// TwinCAT 3 PLC project Abschervorrichtung
// ProgramVersion: 3.1.4026.16
// libraries:
//   Tc2_EtherCAT, * (Beckhoff Automation GmbH)
//   Tc2_Standard, * (Beckhoff Automation GmbH)
//   Tc2_System, * (Beckhoff Automation GmbH)
// project tree:
//   DUTs/ ST_OperatingTime.TcDUT, ST_OpMode.TcDUT (not stored)
//   GVLs/ GVL_CouplerOnDesk.TcGVL (not stored)
//   / PlcTask.TcTTO
//   POUs/ FB_EL6090.TcPOU (not stored), FB_SetOpMode.TcPOU (not stored), F_Convert_to_OperatingTime.TcPOU (not stored), MAIN.TcPOU (not stored), MAIN_1.TcPOU
// real-time tasks:
//   TASK PlcTask: cycle T#10ms, priority 20, ADS port 352
// I/O:
//   DEVICE Master (EtherCAT), AmsNetId 192.168.10.102.2.1
//     Term 1 (EK1101) [EK1101 EtherCAT Coupler (2A E-Bus, ID switch)]
//       Digital Input (EL1014) [EL1014 4Ch. Dig. Input 24V, 10µs]
//       Digital Output (EL2004) [EL2004 4Ch. Dig. Output 24V, 0.5A]
//       Analog Input (EL3064) [EL3064 4Ch. Ana. Input 0-10V]
//       Analog Output (EL4102) [EL4102 2Ch. Ana. Output  0-10V, 16bit]
//       Display (EL6090) [EL6090 Display terminal]
//       Endcover (EL9011) [EL9011 End Terminal]
// variable links:
//   (this object) <-> Master (EtherCAT)
//     PlcTask Inputs/GVL_CouplerOnDesk.bHotConnectGrpState <-> SyncUnits/[DeskGroup]/PlcTask/InfoData/State
//     PlcTask Inputs/GVL_CouplerOnDesk.bHotConnectGrpWcState <-> SyncUnits/[DeskGroup]/PlcTask/InfoData/State
//     PlcTask Inputs/GVL_CouplerOnDesk.nEtherCatDevState <-> Inputs/DevState
//   (this object) <-> Master (EtherCAT)/Term 1 (EK1101)
//     PlcTask Inputs/GVL_CouplerOnDesk.nCouplerId <-> ID/ID
//   (this object) <-> Master (EtherCAT)/Term 1 (EK1101)/Analog Input (EL3064)
//     PlcTask Inputs/GVL_CouplerOnDesk.nPotentiomerValue <-> AI Standard Channel 1/Value
//   (this object) <-> Master (EtherCAT)/Term 1 (EK1101)/Analog Output (EL4102)
//     PlcTask Outputs/GVL_CouplerOnDesk.nPotentiometerSupply <-> Channel 1/Output
//   (this object) <-> Master (EtherCAT)/Term 1 (EK1101)/Digital Input (EL1014)
//     PlcTask Inputs/GVL_CouplerOnDesk.bSelectorSwitch <-> Channel 1/Input
//     PlcTask Inputs/GVL_CouplerOnDesk.bSelectorSwitchLeftNC <-> Channel 2/Input
//     PlcTask Inputs/GVL_CouplerOnDesk.bSelectorSwitchRightNC <-> Channel 3/Input
//   (this object) <-> Master (EtherCAT)/Term 1 (EK1101)/Digital Output (EL2004)
//     PlcTask Outputs/GVL_CouplerOnDesk.bSelectorSwitchLed <-> Channel 1/Output
//   (this object) <-> Master (EtherCAT)/Term 1 (EK1101)/Display (EL6090)
//     PlcTask Inputs/GVL_CouplerOnDesk.bNavDown <-> DIS Inputs/Down
//     PlcTask Inputs/GVL_CouplerOnDesk.bNavEnter <-> DIS Inputs/Enter
//     PlcTask Inputs/GVL_CouplerOnDesk.bNavLeft <-> DIS Inputs/Left
//     PlcTask Inputs/GVL_CouplerOnDesk.bNavRight <-> DIS Inputs/Right
//     PlcTask Inputs/GVL_CouplerOnDesk.bNavUp <-> DIS Inputs/Up
//     PlcTask Inputs/MAIN_1.EL6090_State <-> InfoData/State
//     PlcTask Inputs/MAIN_1.SlaveNetID <-> InfoData/AdsAddr/netId
//     PlcTask Inputs/MAIN_1.SlavePort <-> InfoData/AdsAddr/port
//     PlcTask Outputs/GVL_CouplerOnDesk.nDisplayRow1 <-> DIS Outputs/Value row 1
//     PlcTask Outputs/GVL_CouplerOnDesk.nDisplayRow2 <-> DIS Outputs/Value row 2

CONFIGURATION Abschervorrichtung
    RESOURCE PLC ON TwinCAT3
        TASK PlcTask(INTERVAL := T#10ms, PRIORITY := 20);
        PROGRAM MAIN WITH PlcTask : MAIN;
    END_RESOURCE
END_CONFIGURATION

// ---- DUTs/ST_OperatingTime.TcDUT
TYPE ST_OperatingTime :
STRUCT
	nSec	: INT;
	nMin	: INT;
	nHours	: INT;
	nDays	: INT;
END_STRUCT
END_TYPE

// ---- POUs/MAIN_1.TcPOU
PROGRAM MAIN_1
VAR
	(* Visu Elements*)
	sLine1				:STRING := 'Hello';
	sLine2				:STRING := 'Beckhoff';

	(* Linked Varaibles *)
	SlavePort  AT %I* 	: WORD;
	SlaveNetID AT %I* 	: T_AmsNetIdArr;

	fbTrig				: R_TRIG;
	M_1					: BOOL;
	fb_EL6090			: FB_EL6090;

	StrTime				: ST_OperatingTime;

	EL6090_State AT %I*	: WORD;
END_VAR

IF EL6090_State=16#8 THEN
	fb_EL6090.bAutoUpdate:=TRUE;
END_IF


fb_EL6090(bAutoUpdate:=,
		AmsNetId:=F_CreateAmsNetId(SlaveNetId),
		Port:=SlavePort);
StrTime:=f_Convert_to_OperatingTime(fb_EL6090.nOpertingTime);


(* pos. trig from NAVI "ENTER"*)
fbTrig(CLK:=GVL_CouplerOnDesk.bNavEnter);
IF fbTrig.Q THEN
	M_1:=NOT M_1;
	GVL_CouplerOnDesk.nDisplayRow1:=GVL_CouplerOnDesk.nDisplayRow1+1;
END_IF

GVL_CouplerOnDesk.nDisplayRow2:=GVL_CouplerOnDesk.nDisplayRow2+1;

IF M_1 THEN
	fb_EL6090.strLine_1:=sLine1;
	fb_EL6090.strLine_2:=sLine2;
ELSE
	fb_EL6090.strLine_1:='Value 1:%i';
	fb_EL6090.strLine_2:='Value 2:%i';
END_IF

END_PROGRAM
